{attribute 'linkalways'} 
{attribute 'no_explicit_call' := 'This FB is a CLASS and must be accessed using methods or properties'}
{attribute 'enable_dynamic_creation'}
FUNCTION_BLOCK _TcVnParamsAKAZE EXTENDS StructuredDatatypeBase
VAR
	localData : TcVnParamsAKAZE;
	activeData : REFERENCE TO TcVnParamsAKAZE REF= localData;
    _eDescrType     : _ETcVnFeatureDescriptorTypeAKAZE(localdata.eDescrType);
    _nDescrSize     : _UDINT(localdata.nDescrSize);
    _nDescrChannels : _UDINT(localdata.nDescrChannels);
    _fThreshold     : _REAL(localdata.fThreshold);
    _nOctaves       : _UDINT(localdata.nOctaves);
    _nOctaveLayers  : _UDINT(localdata.nOctaveLayers);
    _eDiffusivity   : _ETcVnDiffusivityTypeKAZE(localdata.eDiffusivity);
END_VAR

PROPERTY PUBLIC Address : PVOID
GET
Address := ADR(activeData);
END_GET
END_PROPERTY

METHOD PUBLIC ClearReference
VAR_INPUT
END_VAR
activeData REF= localData;
SetMemberReference();
END_METHOD

METHOD PUBLIC Clone : I_Datatype
VAR
    pClone : POINTER TO _TcVnParamsAKAZE;
END_VAR
pClone := __NEW(_TcVnParamsAKAZE());
pClone^.Value := Value;
Clone := pClone^;
END_METHOD

PROPERTY PUBLIC eDescrType : REFERENCE TO _ETcVnFeatureDescriptorTypeAKAZE
GET
eDescrType REF= _eDescrType;
END_GET
END_PROPERTY

PROPERTY PUBLIC eDiffusivity : REFERENCE TO _ETcVnDiffusivityTypeKAZE
GET
eDiffusivity REF= _eDiffusivity;
END_GET
END_PROPERTY

METHOD FB_init : BOOL
VAR_INPUT
	bInitRetains : BOOL; // if TRUE, the retain variables are initialized (warm start / cold start)
	bInCopyCode : BOOL;  // if TRUE, the instance afterwards gets moved into the copy code (online change)
END_VAR
SetMemberReference();
AddMember('eDescrType', _eDescrType);
AddMember('nDescrSize', _nDescrSize);
AddMember('nDescrChannels', _nDescrChannels);
AddMember('fThreshold', _fThreshold);
AddMember('nOctaves', _nOctaves);
AddMember('nOctaveLayers', _nOctaveLayers);
AddMember('eDiffusivity', _eDiffusivity);
END_METHOD

PROPERTY PUBLIC fThreshold : REFERENCE TO _REAL
GET
fThreshold REF= _fThreshold;
END_GET
END_PROPERTY

PROPERTY PUBLIC Identifier : T_MAXSTRING
GET
Identifier := 'TcVnParamsAKAZE';
END_GET
END_PROPERTY

METHOD PUBLIC MakeReferenceTo
VAR_INPUT
	ReferenceTarget : REFERENCE TO TcVnParamsAKAZE;
END_VAR
activeData REF= ReferenceTarget;
SetMemberReference();
END_METHOD

PROPERTY PUBLIC nDescrChannels : REFERENCE TO _UDINT
GET
nDescrChannels REF= _nDescrChannels;
END_GET
END_PROPERTY

PROPERTY PUBLIC nDescrSize : REFERENCE TO _UDINT
GET
nDescrSize REF= _nDescrSize;
END_GET
END_PROPERTY

PROPERTY PUBLIC nOctaveLayers : REFERENCE TO _UDINT
GET
nOctaveLayers REF= _nOctaveLayers;
END_GET
END_PROPERTY

PROPERTY PUBLIC nOctaves : REFERENCE TO _UDINT
GET
nOctaves REF= _nOctaves;
END_GET
END_PROPERTY

METHOD PROTECTED SetMemberReference
VAR_INPUT
END_VAR
_eDescrType.MakeReferenceTo(activeData.eDescrType);
_nDescrSize.MakeReferenceTo(activeData.nDescrSize);
_nDescrChannels.MakeReferenceTo(activeData.nDescrChannels);
_fThreshold.MakeReferenceTo(activeData.fThreshold);
_nOctaves.MakeReferenceTo(activeData.nOctaves);
_nOctaveLayers.MakeReferenceTo(activeData.nOctaveLayers);
_eDiffusivity.MakeReferenceTo(activeData.eDiffusivity);
END_METHOD

PROPERTY PUBLIC Size : UDINT
GET
Size := SIZEOF(activeData);
END_GET
END_PROPERTY

METHOD TryMakeReferenceTo : BOOL
VAR_INPUT
	Target : I_Datatype;
END_VAR
VAR
	pTargetData : POINTER TO TcVnParamsAKAZE;
END_VAR
IF NOT IsEquivalentTo(Target) THEN
	RETURN;
END_IF

pTargetData := Target.Address;
activeData REF= pTargetData^;
SetMemberReference();
TryMakeReferenceTo := TRUE;
END_METHOD

PROPERTY PUBLIC Value : REFERENCE TO TcVnParamsAKAZE
GET
Value REF= activeData;
END_GET
END_PROPERTY

END_FUNCTION_BLOCK

(* stored: Version 1.1.0.1, ProductVersion 3.1.4024.13
   POU _TcVnParamsAKAZE: Id {c839a775-c51a-06ec-228a-0ba84390686f}, SpecialFunc None
   Folder Core: Id {1dd5d73a-b6ca-0c17-33a4-98bcae87b5e5}
   Folder Customize: Id {64fe8001-c391-08e1-1fa5-8443ab2fa342}
   Folder Constructor: Id {f237055a-0387-0b84-10a6-bca0af29420f}
   Folder Protected: Id {6edf3c58-ccfd-038c-2108-36d9da898ed8}
   Property Address: Id {bbe65fd1-f93c-0324-011d-65f58e94dbe3}
   Get Get: Id {46724954-455e-0e6e-0f7a-cd44b55146d7}
   Method ClearReference: Id {1e3eefb9-b8f8-00ae-0b15-1971d78c9ff5}
   Method Clone: Id {d7e8744a-eb81-0731-0276-8f730d2f5c80}
   Property eDescrType: Id {4eddb42b-b718-07a4-347d-048b5a772ae5}
   Get Get: Id {7eb7c4d9-231f-0beb-2b9b-54aa0f4dd998}
   Property eDiffusivity: Id {32316acc-0720-04f7-1e89-c8680a7b7257}
   Get Get: Id {faabd0f1-3260-046e-3d9c-6e8f0d60412c}
   Method FB_init: Id {453b60ac-0854-04dc-1f4b-89e927518407}
   Property fThreshold: Id {875f389b-0649-0f99-2382-d6327cddb3e6}
   Get Get: Id {071191ac-3ef0-0603-301d-ce5dca363158}
   Property Identifier: Id {bced6ffe-3c4b-08a2-2173-ef20412b3d4b}
   Get Get: Id {b56f2570-344c-0459-2077-618e97307c08}
   Method MakeReferenceTo: Id {b42cf220-24ec-0235-37b0-605e6305b361}
   Property nDescrChannels: Id {0f7c11a2-6016-09a8-16aa-3ad2ec8d498a}
   Get Get: Id {6bcce512-3f40-0018-1882-6375eda9c8fa}
   Property nDescrSize: Id {d6659a2e-0da5-0916-2f02-649a622738dc}
   Get Get: Id {b4b42b53-6b4e-0827-0f4f-876a116b3db3}
   Property nOctaveLayers: Id {716686a7-0ca3-0153-11cf-fca2155aa4b2}
   Get Get: Id {859ef79a-b786-0f1a-0510-e5c71aa00d7c}
   Property nOctaves: Id {a7cb2d6b-600b-095b-1ec3-2bbb674cf981}
   Get Get: Id {7a8430b8-988c-01e7-0b7d-4bd3ec2c4776}
   Method SetMemberReference: Id {c195b46c-e131-0f28-06c1-694a76f08381}
   Property Size: Id {a14a3206-ac1e-0ef2-0b0f-b17c332e7fbc}
   Get Get: Id {b7f3075a-68e8-0e77-24ba-cde4039f232d}
   Method TryMakeReferenceTo: Id {ab11752d-e4cc-078b-128c-5156b9548b5d}
   Property Value: Id {22af1cae-b476-0eb9-031a-fc870b893c27}
   Get Get: Id {653d7a55-bae9-008a-2b4b-4d1feb2c00d2} *)
